// TIA Portal V20 export
DATA_BLOCK "Instance_FB_IO_Device_Production_And_Rework_DB"   // DB105
// stored: AutoNumber false, InstanceOfName FB_IO_Device_Production_And_Rework, InstanceOfType FB
"FB_IO_Device_Production_And_Rework"
   // VAR_INPUT
   //    Start : Bool;
   //    Manual_Turn_On_Motor_Caroussel : Bool;
   //    Manual_Turn_On_Motor_Conveyor_Belt : Bool;
   //    Water_Foutain_Fail_Functional_Test : Bool;
   //    Select_Motor_Speed : SInt;
   //    Carousel_Voltage_Selection : SInt;
   //    In_PLC_Production_And_Rework : "IO_Device_Conveyor_Belt_Input";
   // END_VAR
   // VAR_OUTPUT
   //    Comunication_Error : Bool;
   //    Emergency_Stop_Release : Bool;
   //    Trigger_Read_Serial_Number_Entrace_Functional_Test : Bool;
   //    Trigger_Read_Serial_Number_Exit_Functional_Test : Bool;
   //    Selected_Voltage_220V : Bool;
   //    Selected_Voltage_127V : Bool;
   //    Carousel_Frequency_Inverter_Fail : Bool;
   //    Conveyor_Belt_Functional_Test_Inverter_Fail : Bool;
   //    Out_PLC_Production_And_Rework : "IO_Device_Conveyor_Belt_Ouput";
   // END_VAR
   // VAR
   //    Timer_Alarme_A_1 { S7_SetPoint := 'True'} : TON_TIME;
   //    Timer_Alarme_B_1 { S7_SetPoint := 'True'} : TON_TIME;
   // END_VAR
BEGIN
END_DATA_BLOCK
